	        ELSIF (#instHome.Error = TRUE) THEN
	          // Errorhandling
	          #statStatus := #ERR_MC_HOME;
	          #statErrorAutoCleared := TRUE;
	          #statDiagnostics.subfunctionStatus := #statSubfunctionStatus := #instHome.ErrorId;
	          #statPassiveHomingState := #NO_HOMING_ACTIVE;
	          // Set next state
	          #statFBState := #AXIS_STOP_ON_ERROR_SELECTION;
	        ELSE
	          ; // Command selected
	        END_IF;
	        #statExeOfHoming := 16#0;
	        #statExeOfHoming.%X0 := #instHome.Busy;
	        #statExeOfHoming.%X1 := #instHome.Done;
	        #statExeOfHoming.%X2 := #instHome.CommandAborted;
	        #statExeOfHoming.%X3 := #instHome.Error;
	      END_REGION
	    ELSE
	      // Errorhandling
	      #statStatus := #ERR_INVALID_HOMING_EXTENDED_MODE;
	      #statErrorAutoCleared := TRUE;
	      #statDiagnostics.subfunctionStatus := #statSubfunctionStatus := 0;
	      #statDiagnostics.basicMotionState := #statBasicMotionState;
	      #statDiagnostics.superimposedMotionState := #statSupImpMotionState;
	      // Set next state
	      #statFBState := #AXIS_STOP_ON_ERROR_SELECTION;
	      #statBasicMotionState := #NO_SELECTION;
	      #statPassiveHomingState := #NO_HOMING_ACTIVE;
	  END_CASE;
	END_REGION

	//----------------------------------------------------------------------------------------------
	// Execution of functionalities of superimposed coordinate system
	//----------------------------------------------------------------------------------------------
	REGION EXECUTION_OF_SUPERIMPOSED_COMMANDS
	  // Statemachine for superimposed motion commands
	  // Write diagnostics
	  #statDiagnostics.basicMotionState := #statBasicMotionState;
	  #statDiagnostics.superimposedMotionState := #statSupImpMotionState;

	  CASE #statSupImpMotionState OF
	    #NO_SELECTION:
	      ; // Do nothing

	    #POS_SUPERIMPOSED_SELECTED:
	      // Additional features (applicative) : Specified direction
	      REGION POS_SUPERIMPOSED_SELECTED;
	        // Firstcycle of command
	        IF (#statFirstCycleSupImpMotion = TRUE) THEN
	          // Configurate the direction of rotation
	          IF ((#configuration.posSuperimposed.direction = 0) AND (#configuration.posSuperimposed.distance >= 0.0))  // Sign of distance is evaluated
	            OR (#configuration.posSuperimposed.direction = #FORWARD_DIR)// Positive direction
	          THEN
	            #statSupImpMotionPosition := ABS(IN := #configuration.posSuperimposed.distance);
	            // Reset MC_MOVESUPERIMPOSED command
	            #instMoveSuperimposed(Axis := #axis,
	                                  Execute := FALSE);
	            #statApplicativeSupImpMotionError := FALSE;
	          ELSIF ((#configuration.posSuperimposed.direction = 0) AND (#configuration.posSuperimposed.distance < 0.0)) // Sign of distance is evaluated
	            OR (#configuration.posSuperimposed.direction = #BACKWARD_DIR)// Negative direction
	          THEN
	            #statSupImpMotionPosition := - ABS(IN := #configuration.posSuperimposed.distance);
	            // Reset MC_MOVESUPERIMPOSED command
	            #instMoveSuperimposed(Axis := #axis,
	                                  Execute := FALSE);
	            #statApplicativeSupImpMotionError := FALSE;
	          ELSE
	            // Errorhandling - Invalid direction
	            #statStatus := #ERR_INVALID_POS_SUPERIMPOSED_DIR;
	            #statErrorAutoCleared := TRUE;
	            #statDiagnostics.subfunctionStatus := #statSubfunctionStatus := 0;
	            #statApplicativeSupImpMotionError := TRUE;
	            // Set next state
	            #statFBState := #AXIS_STOP_ON_ERROR_SELECTION;
	            #statSupImpMotionState := #NO_SELECTION;
	          END_IF;
	        END_IF;

	        IF (#statApplicativeSupImpMotionError = FALSE) THEN
	          // Call MC_Command
	          #instMoveSuperimposed(Axis := #axis,
	                                Execute := #statSupImpCommand.%X0, // Input: posSuperimposed
	                                Distance := #statSupImpMotionPosition,
	                                VelocityDiff := #configuration.posSuperimposed.velocityDiff,
	                                Acceleration := #configuration.posSuperimposed.acceleration,
	                                Deceleration := #configuration.posSuperimposed.deceleration,
	                                Jerk := #configuration.posSuperimposed.jerk);

	          // Evaluate MC_Command
	          IF (#instMoveSuperimposed.Busy = FALSE) AND
	            (#instMoveSuperimposed.Error = FALSE) AND
	            (#instMoveSuperimposed.Done = FALSE) AND
	            (#instMoveSuperimposed.CommandAborted = FALSE)
	          THEN
	            // Return to NO_SELECTION if command finished
	            #statSupImpMotionState := #NO_SELECTION;

	          ELSIF (#instMoveSuperimposed.Error = TRUE) THEN
	            // Errorhandling
	            #statStatus := #ERR_MC_MOVESUPERIMPOSED;
	            #statErrorAutoCleared := TRUE;
	            #statDiagnostics.subfunctionStatus := #statSubfunctionStatus := #instMoveSuperimposed.ErrorId;
	            // Set next state
	            #statFBState := #AXIS_STOP_ON_ERROR_SELECTION;
	            #statSupImpMotionState := #NO_SELECTION;
	          ELSE
	            ; // command selected
	          END_IF;
	          #statExeOfSupImpMotionState := 16#0;
	          #statExeOfSupImpMotionState.%X0 := #instMoveSuperimposed.Busy;
	          #statExeOfSupImpMotionState.%X1 := #instMoveSuperimposed.Done;
	          #statExeOfSupImpMotionState.%X2 := #instMoveSuperimposed.CommandAborted;
	          #statExeOfSupImpMotionState.%X3 := #instMoveSuperimposed.Error;
	        END_IF;
	      END_REGION

	    ELSE
	      // Errorhandling
	      #statStatus := #ERR_UNDEFINED_SUPERIMPOSED_MOTION_STATE;
	      #statErrorUserCleared := TRUE;
	      #statDiagnostics.subfunctionStatus := #statSubfunctionStatus := 0;
	      // Set errorstate
	      #statFBState := #FB_ERROR;
	  END_CASE;
	END_REGION

	//----------------------------------------------------------------------------------------------
	// Execution of torquelimiting functionality
	//----------------------------------------------------------------------------------------------
	REGION EXECUTION_OF_TORQUELIMTING
	  // Statemachine for torquelimiting
	  REPEAT
	    #tempStateChangeActive := FALSE;
	    CASE #statTorqueLimitingState OF
	      #NO_TORQUE_LIMITING_ACTIVE:
	        ;

	      #TORQUE_LIMITING_DISABLE:
	        // Torquelimiting disable
	        #instTorqueLimiting(Axis := #axis,
	                            Enable := FALSE);

	        // Check state of torque limting
	        IF (#instTorqueLimiting.Busy = FALSE)
	        THEN
	          // set next state
	          #statTorqueLimitingState := #NO_TORQUE_LIMITING_ACTIVE;
	        ELSE
	          ; // Waiting for MC_Torquelimiting is not busy
	        END_IF;

	      #TORQUE_LIMTING_SELECTED:
	        // No extended homing function active
	        #instTorqueLimiting(Axis := #axis,
	                            Enable := #statExtendedCommand.%X1,
	                            Limit := #configuration.torqueLimiting.limit,
	                            Mode := #configuration.torqueLimiting.mode);

	        IF (#instTorqueLimiting.Busy = FALSE) THEN
	          // Reset state
	          #statTorqueLimitingState := #NO_TORQUE_LIMITING_ACTIVE;
	        END_IF;

	      #FIXED_STOP_DETECTION_ACTIVE:
	        // Extended homing function active
	        #instTorqueLimiting(Axis := #axis,
	                            Enable := TRUE,
	                            Limit := #configuration.homing.extendedModeTorqueLimit, // V01.00.03 Always use configured value
	                            Mode := #MODE_FIXED_STOP_DETECTION);

	        IF ((#statHomingSubState = #HOMING_IDLE) AND (#statBasicMotionState = #ACTIVE_HOMING_SELECTED))
	        THEN
	          // Fixed stop process has finished - Axis is still in clamping
	          #statTorqueLimitingState := #FIXED_STOP_DETECTION_FINISHED;
	          #tempStateChangeActive := TRUE;

	        ELSIF (#statBasicMotionState <> #ACTIVE_HOMING_SELECTED)
	        THEN
	          // Error occurred - change state depending on inClamping
	          IF (#instTorqueLimiting.InClamping = TRUE)
	          THEN
	            // Axis is in clamping
	            #statTorqueLimitingState := #FIXED_STOP_DETECTION_ERROR_IN_CLAMPING;
	            #tempStateChangeActive := TRUE;
	          ELSE
	            // Axis is in not clamping
	            #statTorqueLimitingState := #FIXED_STOP_DETECTION_ERROR_NOT_IN_CLAMPING;
	            #tempStateChangeActive := TRUE;
	          END_IF;
	        ELSE
	          ; // Fixed stop detection is running
	        END_IF;

	      #FIXED_STOP_DETECTION_FINISHED:
	        // Homing on fixed stop process has finished
	        #instTorqueLimiting(Axis := #axis,
	                            Enable := TRUE,
	                            Limit := #configuration.homing.extendedModeTorqueLimit, // V01.00.03 Always use configured value
	                            Mode := #MODE_FIXED_STOP_DETECTION);

	        IF (#instTorqueLimiting.InClamping = FALSE)
	        THEN
	          // InClamping = FALSE
	          IF (#statExtendedCommand.%X1 = TRUE) // Torquelimiting
	          THEN
	            #statTorqueLimitingState := #TORQUE_LIMTING_SELECTED;
	          ELSE
	            #statTorqueLimitingState := #TORQUE_LIMITING_DISABLE;
	          END_IF;
	          #tempStateChangeActive := TRUE;
	        ELSE
	          // InClamping = TRUE
	          IF (#statExtendedCommand.%X1 = TRUE) // Torquelimiting
	            AND (#configuration.torqueLimiting.mode = #MODE_FIXED_STOP_DETECTION)
	          THEN
	            // Change State
	            #statTorqueLimitingState := #TORQUE_LIMTING_SELECTED;
	            #tempStateChangeActive := TRUE;
	          ELSE
	            ; // Wait for inClamping = FALSE
	          END_IF;
	        END_IF;

	      #FIXED_STOP_DETECTION_ERROR_IN_CLAMPING:
	        // Errorstate, torquelimiting is still active and axis not in clamping
	        #instTorqueLimiting(Axis := #axis,
	                            Enable := TRUE,
	                            Limit := #configuration.homing.extendedModeTorqueLimit, // V01.00.03 Always use configured value
	                            Mode := #MODE_FIXED_STOP_DETECTION);

	        IF (#instTorqueLimiting.InClamping = FALSE)
	        THEN
	          // InClamping = FALSE -> reset torque limiting state
	          #statTorqueLimitingState := #TORQUE_LIMITING_DISABLE;
	          // Torquelimiting disable
	          #tempStateChangeActive := TRUE;
	        END_IF;

	      #FIXED_STOP_DETECTION_ERROR_NOT_IN_CLAMPING:
	        // Errorstate, torquelimiting is still active and axis in clamping
	        #instTorqueLimiting(Axis := #axis,
	                            Enable := TRUE,
	                            Limit := #configuration.homing.extendedModeTorqueLimit, // V01.00.03 Always use configured value
	                            Mode := #MODE_FIXED_STOP_DETECTION);

	        IF (#instTorqueLimiting.InClamping = TRUE)
	        THEN
	          // InClamping = TRUE -> change state
	          #statTorqueLimitingState := #FIXED_STOP_DETECTION_ERROR_IN_CLAMPING;
	          #tempStateChangeActive := TRUE;

	        ELSIF (#statBasicMotionState <> #NO_SELECTION)
	          OR (#statSupImpMotionState <> #NO_SELECTION)
	          OR (#statPassiveHomingState <> #NO_HOMING_ACTIVE)
	        THEN
	          // New valid command is set -> reset error state
	          #statTorqueLimitingState := #TORQUE_LIMITING_DISABLE;
	          #tempStateChangeActive := TRUE;
	        ELSE
	          ; // Waiting for new command or axis is getting in clamping
	        END_IF;
	      ELSE
	        // Errorhandling
	        #statStatus := #ERR_UNDEFINED_TORQUE_LIMITING_STATE;
	        #statErrorUserCleared := TRUE;
	        #statDiagnostics.basicMotionState := #statBasicMotionState;
	        #statDiagnostics.superimposedMotionState := #statSupImpMotionState;
	        #statDiagnostics.subfunctionStatus := #statSubfunctionStatus := 0;
	        // Set errorstate
	        #statFBState := #FB_ERROR;
	    END_CASE;
	  UNTIL (#tempStateChangeActive = FALSE)
	  END_REPEAT;
	  // Evaluate MC_Command
	  IF (#instTorqueLimiting.Error = TRUE) AND ((#statTorqueLimitingErrorOld = FALSE) OR (#statStatus = #STATUS_SUBSEQUENT_CALL)) THEN
	    // Errorhandling
	    #statStatus := #ERR_MC_TORQUELIMITING;
	    #statErrorAutoCleared := TRUE;
	    #statDiagnostics.basicMotionState := #statBasicMotionState;
	    #statDiagnostics.superimposedMotionState := #statSupImpMotionState;
	    #statDiagnostics.subfunctionStatus := #statSubfunctionStatus := #instTorqueLimiting.ErrorId;

	    #statFBState := #AXIS_STOP_ON_ERROR_SELECTION;

	  ELSIF (#instTorqueLimiting.Error = FALSE) AND ((#statTorqueLimitingErrorOld = TRUE) AND (#statStatus = #ERR_MC_TORQUELIMITING)) THEN
	    #statStatus := #STATUS_SUBSEQUENT_CALL;
	    #statErrorAutoCleared := FALSE;
	  ELSE
	    ;
	  END_IF;

	  #statTorqueLimitingErrorOld := #instTorqueLimiting.Error;
	END_REGION

	//----------------------------------------------------------------------------------------------
	// Selection of StopOnError / implementation of fastStop
	//----------------------------------------------------------------------------------------------
	REGION STOP_ON_ERROR
	  // Check for stopping if error occurred during execution of motion commands
	  IF (#statFBState = #AXIS_STOP_ON_ERROR_SELECTION)
	  THEN
	    #statBasicMotionState := #NO_SELECTION;
	    #statSupImpMotionState := #NO_SELECTION;
	    #statPassiveHomingState := #NO_HOMING_ACTIVE;

	    IF (#configuration.generalSettings.stopOnError = TRUE)
	    THEN
	      // Read Statusword
	      #tempStatusWord := #axis.StatusWord;

	      // Evaluate error
	      IF #tempStatusWord.%X0 THEN
	        // Axis enabled
	        IF (#tempStatusWord.%X1 = TRUE) THEN
	          // TO Alarm present
	          #statFBState := #AXIS_MOTION;
	        ELSE
	          // No TO alarm present, set fastStop
	          //#statBasicMotionState := #FAST_STOP_SELECTED; // V1.1.0
	          #statStopWithoutSignalization := TRUE; // V1.1.0
	          #statFirstCycleBasicMotion := TRUE;
	          #statFBState := #AXIS_STOP_ON_ERROR_EXECUTION;
	        END_IF;
	      ELSE
	        // Axis disabled
	        #statFBState := #AXIS_MOTION;
	      END_IF;
	    ELSE
	      // Dont StopOnError
	      #statFBState := #AXIS_MOTION;
	    END_IF;
	  END_IF;

	  // Implementation of fastStop
	  IF (#statBasicMotionState = #FAST_STOP_SELECTED)
	    OR #statStopWithoutSignalization
	  THEN
	    // Additional feature: Load emergency stop dynamics (TO) if no valid dynamics are configured for fastStop
	    REGION FASTSTOP SELECTED
	      // Firstcycle of command
	      IF (#statFirstCycleBasicMotion = TRUE) THEN
	        // Reset HALT command
	        #instHalt(Axis := #axis,
	                  Execute := FALSE);
	        #statFirstCycleDone := TRUE;
	        // Check dynamics for fastStop
	        // Load TO emergency Stop dynamics if value <=0 for deceleration is configured
	        IF (#configuration.fastStop.deceleration <= 0.0) // V1.0.2 Read TO emergencyStop deceleration only if fastStop.deceleration <= 0
	        THEN
	          // Invalid fastStop dynamics configured - read emergency stop dynamics from TO
	          #statDeceleration := #axis.DynamicDefaults.EmergencyDeceleration;
	        ELSE
	          // Valid fastStop dynamics configured
	          #statDeceleration := #configuration.fastStop.deceleration;
	        END_IF;
	        #statJerk := #configuration.fastStop.jerk; // V1.0.2 Use always configuration for jerk value
	        #statAbortAcceleration := #configuration.fastStop.abortAcceleration; // V1.0.2 Use always configuration
	      END_IF;

	      // Call of MC_Command
	      #instHalt(Axis := #axis,
	                Execute := (#statBasicCommand.%X0 OR #statFirstCycleBasicMotion),
	                Deceleration := #statDeceleration,
	                AbortAcceleration := #statAbortAcceleration,
	                Jerk := #statJerk);

	      // Evaluate MC_Command
	      IF (#instHalt.Busy = FALSE) AND
	        (#instHalt.Error = FALSE) AND
	        (#instHalt.Done = FALSE) AND
	        (#instHalt.CommandAborted = FALSE)
	      THEN
	        // Return to NO_SELECTION if command finished
	        #statFBState := #AXIS_MOTION;
	        #statBasicMotionState := #NO_SELECTION;
	        #statStopWithoutSignalization := FALSE; // V1.1.0

	      ELSIF (#instHalt.Done = TRUE)
	      THEN
	        IF (#statFirstCycleDone = TRUE)
	        THEN
	          // Command is reset
	          IF (#instTorqueLimiting.Error = FALSE) // V1.00.03 Dont reset error is pending
	          THEN
	            // Reset status not if torquelimiting error is pending
	            IF #statStopWithoutSignalization THEN
	              ;
	            ELSE
	              #statStatus := #STATUS_SUBSEQUENT_CALL;
	              #statErrorAutoCleared := FALSE;
	            END_IF;
	          END_IF;

	          #statFirstCycleDone := FALSE;
	        END_IF;
	      ELSE
	        ; // Command selected
	      END_IF;

	      // Write MC_Command outputs to internal variable
	      #statExeOfBasicMotion := 0;
	      #statExeOfBasicMotion.%X0 := #instHalt.Busy;
	      #statExeOfBasicMotion.%X1 := #instHalt.Done;
	      #statExeOfBasicMotion.%X2 := #instHalt.CommandAborted;
	      #statExeOfBasicMotion.%X3 := #instHalt.Error;
	    END_REGION
	  END_IF;
	END_REGION
	//----------------------------------------------------------------------------------------------
	// Store values and reset variables
	//----------------------------------------------------------------------------------------------
	REGION STORE_AND_RESET
	  // Reset variables to determine first cycle of a new command
	  IF (#statFirstCycleReset = TRUE) THEN
	    #statFirstCycleReset := FALSE;
	  END_IF;
	  IF (#statFirstCycleHoming = TRUE) THEN
	    #statFirstCycleHoming := FALSE;
	  END_IF;
	  #statHomingOld := #tempHoming;

	  #statFirstCycleBasicMotion := FALSE;
	  #statBasicCommandOld := #statBasicCommand;

	  IF (#statFirstCycleSupImpMotion = TRUE) THEN
	    #statFirstCycleSupImpMotion := FALSE;
	  END_IF;
	  #statSupImpCommandOld := #statSupImpCommand;

	  // Store last values for edge detection
	  #statEnableOld := #tempEnable;
	  #statEnableAxisOld := #tempEnableAxis;
	  #statExtendedCommandOld := #statExtendedCommand;
	  #statPowerErrorOld := #instPower.Error;
	END_REGION

	//----------------------------------------------------------------------------------------------
	// Writing outputs
	//----------------------------------------------------------------------------------------------
	REGION WRITING_OF_OUTPUTS
	  // Writing status outputs
	  #resetActive := (#statResetState = #CMD_BUSY);

	  IF (#statErrorUserCleared = TRUE) THEN
	    ; // Reset variables at ErrorUserCleared
	    #statBasicMotionState := #NO_SELECTION;
	    #statExeOfBasicMotion := #NO_SELECTION;
	    #statSupImpMotionState := #NO_SELECTION;
	    #statExeOfSupImpMotionState := #NO_SELECTION;
	    #statExeOfHoming := #NO_SELECTION;
	  END_IF;
	  IF (#instPower.Status = TRUE)
	  THEN
	    // Axis enabled
	    #axisEnabled := TRUE;

	  ELSIF (#instPower.Error = TRUE) AND (#instPower.Status = FALSE)
	  THEN
	    // Reset status if error occurred
	    #axisEnabled := FALSE;

	  ELSIF (#instPower.Busy = FALSE)
	  THEN
	    // Reset if MC_Power is not busy
	    #axisEnabled := FALSE;
	  ELSE
	    ;
	  END_IF;

	  REGION WRITING_BASICMOTION_OUTPUTS
	    // Writing Busy, Done and Aborted outputs for basic motion commands
	    IF (#statBasicMotionState > #NO_SELECTION) AND (#statBasicMotionState < #ACTIVE_HOMING_SELECTED)
	    THEN
	      #commandBusy := #statExeOfBasicMotion.%X0;
	      #commandDone := #statExeOfBasicMotion.%X1;
	      #commandAborted := #statExeOfBasicMotion.%X2;
	      #inVelocity := #statExeOfBasicMotion.%X4;
	    ELSE
	      #commandBusy := FALSE;
	      #commandDone := FALSE;
	      #commandAborted := FALSE;
	      #inVelocity := FALSE;
	    END_IF;

	    // Writing outputs up to LAxisCtrl_SpeedAxis
	    IF (#statTorqueLimitingState = #TORQUE_LIMTING_SELECTED)
	      // OR (#statTorqueLimitingState = #AUTOMATIC_MODE_CHANGE) V1.0.3 TorqueLimtinig = TRUE, only when respective value used
	    THEN
	      #torqueLimitingSelected := TRUE;
	    ELSE
	      #torqueLimitingSelected := FALSE;
	    END_IF;

	    #inLimitation := #instTorqueLimiting.InLimitation;
	    #fastStopSelected := #statBasicMotionState.%X0;
	    #stopSelected := #statBasicMotionState.%X1;
	    #jogSelected := #statBasicMotionState.%X2 OR #statBasicMotionState.%X3;
	    #moveVelocitySelected := #statBasicMotionState.%X4;
	    // Writing outputs up to LAxisCtrl_PosAxis
	    #inClamping := #instTorqueLimiting.InClamping;
	    #posRelativeSelected := #statBasicMotionState.%X5;
	    #posAbsoluteSelected := #statBasicMotionState.%X6;
	  END_REGION
	  REGION WRITING_HOMING_OUTPUTS
	    // Writing Busy, Done and Aborted outputs for homing
	    IF (#statPassiveHomingState = #STANDARD_HOMING)
	    THEN
	      #homingSelected := TRUE;
	      #homingCommandBusy := #statExeOfHoming.%X0;
	      #homingCommandDone := #statExeOfHoming.%X1;
	      #homingCommandAborted := #statExeOfHoming.%X2;
	    ELSE
	      IF (#statBasicMotionState = #ACTIVE_HOMING_SELECTED)
	      THEN
	        #homingSelected := TRUE;
	        #homingCommandBusy := #statExeOfBasicMotion.%X0;
	        #homingCommandDone := #statExeOfBasicMotion.%X1;
	        #homingCommandAborted := #statExeOfBasicMotion.%X2;
	      ELSE
	        #homingSelected := FALSE;
	        #homingCommandBusy := FALSE;
	        #homingCommandDone := FALSE;
	        #homingCommandAborted := FALSE;
	      END_IF;
	    END_IF;
	  END_REGION
	  REGION WRITING_SUPERIMPOSED_OUTPUTS
	    // Writing outputs for superimposed motion commands
	    IF (#statSupImpMotionState <> #NO_SELECTION)
	    THEN
	      #superimposedBusy := #statExeOfSupImpMotionState.%X0;
	      #superimposedDone := #statExeOfSupImpMotionState.%X1;
	      #superimposedAborted := #statExeOfSupImpMotionState.%X2;
	    ELSE
	      #superimposedBusy := FALSE;
	      #superimposedDone := FALSE;
	      #superimposedAborted := FALSE;
	    END_IF;
	    #posSuperimposedSelected := #statSupImpMotionState.%X0;
	  END_REGION
	END_REGION

	//----------------------------------------------------------------------------------------------
	// Error handling
	//----------------------------------------------------------------------------------------------
	REGION ERROR_HANDLING
	  IF #statErrorUserCleared THEN
	    #valid := FALSE;
	    #busy := TRUE;
	    #error := TRUE;
	    #status := #statStatus;
	    #subfunctionStatus := #statSubfunctionStatus; // V1.1.0
	    #statDiagnostics.status := #statStatus;

	  ELSIF #statErrorAutoCleared THEN
	    #valid := FALSE;
	    #busy := TRUE;
	    #error := TRUE;
	    #status := #statStatus;
	    #subfunctionStatus := #statSubfunctionStatus; // V1.1.0
	    #statDiagnostics.status := #statStatus;

	  ELSE
	    // Process normal output values
	    #valid := TRUE;
	    #error := FALSE;
	    #status := #statStatus;
	    #subfunctionStatus := #statSubfunctionStatus := 16#0; // V1.1.0
	  END_IF;

	  #diagnostics := #statDiagnostics; // V1.1.0
	END_REGION
END_FUNCTION_BLOCK

